FUNCTION_BLOCK TSetWindowsClock
VAR
    Execution : TExecution;
    NT_SetLocalTime1 : NT_SetLocalTime;
END_VAR

NT_SetLocalTime1(
	NETID:= , 
	TIMESTR:= , 
	START:= Execution.Starting, 
	TMOUT:= , 
	BUSY=> , 
	ERR=> , 
	ERRID=> );
    
IF Execution.Starting THEN
    Execution.SetBusy();
END_IF

IF Execution.Busy AND NOT NT_SetLocalTime1.BUSY THEN
    IF NT_SetLocalTime1.ERR THEN
        Execution.SetError(ErrorId := NT_SetLocalTime1.ERRID);
    ELSE
        Execution.SetDone();
	END_IF
END_IF

METHOD Execute : BOOL
VAR_INPUT
    AmsNetId : T_AmsNetID;
    TimeStruct : TimeStruct;
END_VAR
IF Execution.Start() THEN
    NT_SetLocalTime1.TIMESTR := TimeStruct;
    NT_SetLocalTime1.NETID := AmsNetId;
    Execute := TRUE;
END_IF
END_METHOD

PROPERTY ExecutionResult  : IExecutionResult
GET
ExecutionResult := Execution;
END_GET
END_PROPERTY

END_FUNCTION_BLOCK

(* stored: Version 1.1.0.1, ProductVersion 3.1.4024.3
   POU TSetWindowsClock: Id {4d1bc0b8-9fe6-0162-2bee-7a57f7345d8c}, SpecialFunc None
   Method Execute: Id {33693459-5f31-092d-2f4f-dbe9fe75b222}
   Property ExecutionResult: Id {50d90d7f-91d9-0fde-341e-05e92f759faf}
   Get Get: Id {3e3a2405-6dfa-05d7-3b45-82ed283c24e3} *)
